Staubli VAL3: decodeConfig.pgx

program decodeConfig(pointRx& value, num& buffer[])
begin
  if buffer[0] == 0
    value.config.shoulder = sfree
  elseIf buffer[0] == 1
    value.config.shoulder = ssame
  elseIf buffer[0] == 2
    value.config.shoulder = righty
  elseIf buffer[0] == 3
    value.config.shoulder = lefty
  endIf

  if buffer[1] == 0
    value.config.elbow = efree
  elseIf buffer[1] == 1
    value.config.elbow = esame
  elseIf buffer[1] == 2
    value.config.elbow = epositive
  elseIf buffer[1] == 3
    value.config.elbow = enegative
  endIf

  if buffer[2] == 0
    value.config.wrist = wfree
  elseIf buffer[2] == 1
    value.config.wrist = wsame
  elseIf buffer[2] == 2
    value.config.wrist = wpositive
  elseIf buffer[2] == 3
    value.config.wrist = wnegative
  endIf

  logMsg("S: " + toString("", buffer[0]) + "  E: " + toString("", buffer[1]) + "  W: " + toString("", buffer[2]))
end
